INTERFACE InterfaceObserverBase

END_INTERFACE

(* stored: Version 1.1.0.1, ProductVersion 3.1.4024.15
   Itf InterfaceObserverBase: Id {57ec505c-9aba-4a5b-af23-bb18b464f7a4} *)
